FUNCTION_BLOCK FB_Subsystem
VAR_INPUT
END_VAR
VAR_OUTPUT
END_VAR
VAR
	iInput : INT;
	iOutput : INT;
END_VAR

IF iInput = 66 THEN
	iOutput := 99;
END_IF

{attribute 'monitoring' := 'variable'}
{attribute 'monitoring' := 'call'}
PROPERTY Input : INT
SET
iInput := Input;
END_SET
END_PROPERTY

{attribute 'monitoring' := 'variable'}
{attribute 'monitoring' := 'call'}
PROPERTY Output : INT
GET
Output := iOutput;
END_GET
END_PROPERTY

END_FUNCTION_BLOCK

(* stored: Version 1.1.0.1, ProductVersion 3.1.4024.12
   POU FB_Subsystem: Id {ab3fc085-c768-42c3-a433-84834ffda54a}, SpecialFunc None
   Property Input: Id {f5dcf4b8-1cd4-4bb2-bd5e-69745bef9350}
   Set Set: Id {f34f6e86-a5d6-4669-9220-0574243f434e}
   Property Output: Id {fde8b9d3-5545-4818-bb59-260b78222f7b}
   Get Get: Id {1d42b521-2931-4dac-9731-d59a54efdaa1} *)
